Fanuc TP program (LS listing): FOLGE020.LS

/PROG  FOLGE020
/ATTR
OWNER		= MNEDITOR;
COMMENT		= "VW336";
PROG_SIZE	= 3396;
CREATE		= DATE 23-07-08  TIME 09:33:28;
MODIFIED	= DATE 23-07-08  TIME 12:51:58;
FILE_NAME	= FOLGE011;
VERSION		= 0;
LINE_COUNT	= 22;
MEMORY_SIZE	= 5932;
PROTECT		= READ_WRITE;
TCD:  STACK_SIZE	= 500,
      TASK_PRIORITY	= 50,
      TIME_SLICE	= 0,
      BUSY_LAMP_OFF	= 0,
      ABORT_REQUEST	= 0,
      PAUSE_REQUEST	= 0;
DEFAULT_GROUP	= 1,1,1,1,*;
CONTROL_CODE	= 00000000 00000000;
/APPL
/MN
   1:  UTOOL_NUM=1 ;
   2:  UFRAME_NUM=0 ;
   3:  PAYLOAD[1] ;
   4:J P[1] 10% CNT0 ACC100 TB   0.00sec,P-SPS    ;
      1:  IF (DO[12]),CALL MAKRO998 ;
      2:  DO[15]=ON ;
      3:  DO[16]=ON ;
      4:  CALL MAKRO000    ;
      5:  WAIT (DI[9])    ;
       ------ ;
   5:J P[2] 100% CNT0 ACC100 TB   0.00sec,P-SPS    ;
      1:  TC_ONLINE (ON) ;
      2:  DO[23]=OFF ;
      3:  TIMER[1]=RESET ;
      4:  TIMER[1]=START ;
      5:  CALL MAKRO050    ;
      6:  !lib. de Herramientas ;
      7:  DO[80]=ON ;
      8:  !Lib. de Anticolisiones ;
      9:  DO[41]=ON ;
     10:  DO[42]=ON ;
     11:  DO[45]=ON ;
     12:  DO[46]=ON ;
     13:  !Apagar Posicion Base ;
     14:  DO[15]=OFF ;
     15:  !Fresado EZ1 ;
     16:  F[298]=(OFF) ;
     17:  CALL VW_USER(Basic1,EZSP,Nr1 Service,ProgNr=31, , ,S-Punkt=31, ,EIN/AUS=1) ;
     18:  WAIT    .10(sec) ;
     19:  F[79]=((DI[786] AND !DI[788]) OR (!DI[788] AND DI[130])) ;
     20:  F[78]=(DI[788] AND !F[79]) ;
     21:  WAIT (DI[23])    ;
     22:  DO[23]=ON ;
     23:  TC_ONLINE (M[30] AND M[95]) ;
       ------ ;
   6:  LBL[1] ;
   7:  IF (F[78] OR F[79] OR F[298]),CALL UP101 ;
   8:  IF (F[298]),JMP LBL[1] ;
   9:  !Llamar a UP001 ;
  10:  !Soldar en estacion de Geometria ;
  11:  ! ST1160 ;
  12:J P[3] 100% CNT0 ACC100 TB    .10sec,P-SPS    ;
      1:  TC_ONLINE (ON) ;
      2:  DO[23]=OFF ;
      3:  WAIT (DI[23])    ;
      4:  DO[23]=ON ;
      5:  TC_ONLINE (M[30] AND M[95]) ;
       ------ ;
  13:  CALL UP021    ;
  14:  UFRAME_NUM=0 ;
  15:  UTOOL_NUM=1 ;
  16:J P[4] 100% CNT0 ACC100 TB    .10sec,P-SPS    ;
      1:  TC_ONLINE (ON) ;
      2:  DO[23]=OFF ;
      3:  !Fresado EZ1 ;
      4:  F[298]=(OFF) ;
      5:  CALL VW_USER(Basic1,EZSP,Nr1 Service,ProgNr=31, , ,S-Punkt=31, ,EIN/AUS=1) ;
      6:  WAIT    .10(sec) ;
      7:  F[79]=((DI[786] AND !DI[788]) OR (!DI[788] AND DI[130])) ;
      8:  F[78]=(DI[788] AND !F[79]) ;
      9:  WAIT (DI[23])    ;
     10:  DO[23]=ON ;
     11:  TC_ONLINE (M[30]) ;
       ------ ;
  17:  LBL[2] ;
  18:  IF (F[78] OR F[79] OR F[298]),CALL UP101 ;
  19:  IF (F[298]),JMP LBL[2] ;
  20:  !Fin de Trabajo Total ;
  21:J P[5] 100% CNT0 ACC100 TB    .10sec,P-SPS    ;
      1:  TC_ONLINE (ON) ;
      2:  DO[23]=OFF ;
      3:  CALL MAKRO015    ;
      4:  WAIT (DI[23])    ;
      5:  DO[23]=ON ;
      6:  TC_ONLINE (M[30]) ;
       ------ ;
  22:J P[6] 100% CNT0 ACC100 TB   0.00sec,P-SPS    ;
      1:  TC_ONLINE (ON) ;
      2:  DO[14]=ON ;
      3:  DO[15]=ON ;
      4:  TIMER[1]=STOP ;
      5:  TIMER[2]=(TIMER[1]) ;
      6:  TIMER[2]=STOP ;
       ------ ;
/POS
P[1]{
   GP1:
	UF : 0, UT : 1,		CONFIG : 'F U T, 0, 1, 0',
	X =  1731.500  mm,	Y =     2.242  mm,	Z =  -321.863  mm,
	W =  -176.060 deg,	P =    33.147 deg,	R =  -172.829 deg
   GP2:
	UF : 0, UT : 1,
	J1=   300.000  mm
   GP3:
	UF : 0, UT : 1,
	J1=     0.000  mm
   GP4:
	UF : 0, UT : 1,
	J1=     0.000  mm
};
P[2]{
   GP1:
	UF : 0, UT : 1,		CONFIG : 'F U T, 0, 1, 0',
	X =  1731.500  mm,	Y =     2.242  mm,	Z =  -321.863  mm,
	W =  -176.060 deg,	P =    33.147 deg,	R =  -172.829 deg
   GP2:
	UF : 0, UT : 1,
	J1=   300.000  mm
   GP3:
	UF : 0, UT : 1,
	J1=     0.000  mm
   GP4:
	UF : 0, UT : 1,
	J1=     0.000  mm
};
P[3]{
   GP1:
	UF : 0, UT : 1,		CONFIG : 'F U T, 0, 1, 0',
	X =  1731.500  mm,	Y =     2.242  mm,	Z =  -321.863  mm,
	W =  -176.060 deg,	P =    33.147 deg,	R =  -172.829 deg
   GP2:
	UF : 0, UT : 1,
	J1=   300.000  mm
   GP3:
	UF : 0, UT : 1,
	J1=     0.000  mm
   GP4:
	UF : 0, UT : 1,
	J1=     0.000  mm
};
P[4]{
   GP1:
	UF : 0, UT : 1,		CONFIG : 'F U T, 0, 1, 0',
	X =  1731.500  mm,	Y =     2.242  mm,	Z =  -321.863  mm,
	W =  -176.060 deg,	P =    33.147 deg,	R =  -172.829 deg
   GP2:
	UF : 0, UT : 1,
	J1=   300.000  mm
   GP3:
	UF : 0, UT : 1,
	J1=     0.000  mm
   GP4:
	UF : 0, UT : 1,
	J1=     0.000  mm
};
P[5]{
   GP1:
	UF : 0, UT : 1,		CONFIG : 'F U T, 0, 1, 0',
	X =  1731.500  mm,	Y =     2.242  mm,	Z =  -321.863  mm,
	W =  -176.060 deg,	P =    33.147 deg,	R =  -172.829 deg
   GP2:
	UF : 0, UT : 1,
	J1=   300.000  mm
   GP3:
	UF : 0, UT : 1,
	J1=     0.000  mm
   GP4:
	UF : 0, UT : 1,
	J1=     0.000  mm
};
P[6]{
   GP1:
	UF : 0, UT : 1,		CONFIG : 'F U T, 0, 1, 0',
	X =  1731.500  mm,	Y =     2.242  mm,	Z =  -321.863  mm,
	W =  -176.060 deg,	P =    33.147 deg,	R =  -172.829 deg
   GP2:
	UF : 0, UT : 1,
	J1=   300.000  mm
   GP3:
	UF : 0, UT : 1,
	J1=     0.000  mm
   GP4:
	UF : 0, UT : 1,
	J1=     0.000  mm
};
/END
